{attribute 'linkalways'} 
{attribute 'no_explicit_call' := 'This FB is a CLASS and must be accessed using methods or properties'}
{attribute 'enable_dynamic_creation'}
FUNCTION_BLOCK Node_F_VN_CreateEmptyImage EXTENDS VisionNode
VAR
    ipImage : _ITcVnImage;
    hrPrev : _HRESULT(S_OK);
	hresult : _HRESULT(S_OK);
END_VAR

METHOD PUBLIC  Clone : I_Node
VAR
	pNode : POINTER TO Node_F_VN_CreateEmptyImage;
END_VAR
pNode := __NEW(Node_F_VN_CreateEmptyImage);
Clone := pNode^;
END_METHOD

METHOD FB_init : BOOL
VAR_INPUT
	bInitRetains : BOOL; // if TRUE, the retain variables are initialized (warm start / cold start)
	bInCopyCode : BOOL;  // if TRUE, the instance afterwards gets moved into the copy code (online change)
END_VAR
AddInput('hrPrev', hrPrev);
AddOutput('ipImage', ipImage);
AddOutput('hresult',hresult);
END_METHOD

METHOD PROTECTED OnExecute
hresult.Value := F_VN_CreateEmptyImage(
    ipImage := ipImage.Value,
	hrPrev:= hrPrev.Value);
END_METHOD

METHOD PUBLIC PreExecutionCheck
VAR_INPUT
	Check : I_PreExecutionChecks;
END_VAR
END_METHOD

END_FUNCTION_BLOCK

(* stored: Version 1.1.0.1, ProductVersion 3.1.4024.13
   POU Node_F_VN_CreateEmptyImage: Id {d5958470-5868-036e-3902-02d760f8e03c}, SpecialFunc None
   Folder Constructor: Id {e3ff68f6-8ebf-0cf1-1cee-9f2201fea929}
   Method Clone: Id {b5953517-7762-0334-19cd-4591e3f6bbea}
   Method FB_init: Id {1122572b-c114-0588-1a9f-765db0d78815}
   Method OnExecute: Id {d615950f-5987-0c78-2d5d-919af1aba5f4}
   Method PreExecutionCheck: Id {c5c3b9ef-03e6-088c-0789-f179001f5045} *)
